TYPE ST_Probes_I_O :
STRUCT
	
	anDistances						: ARRAY[0..5] OF DINT;
	abProbeError					: ARRAY[0..7] OF BOOL;
	bGeneralError					: BOOL;
	anRawMeasurement				: ARRAY[0..7] OF DINT;
	bSetDistances					: BOOL;
	
	
END_STRUCT
END_TYPE

(* stored: Version 1.1.0.1, ProductVersion 3.1.4024.13
   DUT ST_Probes_I_O: Id {84e24643-423a-42da-8153-4f00aca97b7f} *)
